// TIA Portal V20 export
TYPE "typeEmDataControlNode"
// stored: Namespace Unit1.Em7
   STRUCT
      hotPressLeft { S7_SetPoint := 'True'} : "LER_typePartData";
      hotPressRight { S7_SetPoint := 'True'} : "LER_typePartData";
      transferPnPLeft : "LER_typePartData";
      transferPnPRight : "LER_typePartData";
      hipotThickness : "LER_typePartData";
   END_STRUCT;
END_TYPE
